SUBAPPLICATION Uebung_206b_AX (* Interlock: ILOCK_T_FF_SR_AX (2 gegenseitig verriegelte Toggle-Flip-Flops via Adapter-Kette, zusaetzlich direktes Set/Reset auf FF1) *)
  (* Standard: 61499-2; Description: Copyright (c) 2026 Meisterschulen am Ostbahnhof This program and the accompanying materials are made available under the terms of the Eclipse Public License 2.0 which is available at https://www.eclipse.org/legal/epl-2.0/ SPDX-License-Identifier: EPL-2.0 *)
  (* Version 1.0, 2026-09-07, Franz Höpfinger, Meisterschulen am Ostbahnhof, initial API and implementation and/or initial documentation - TRAINING_GAPS.md Punkt 7 *)
  PACKAGE Uebungen;
  IMPORT logiBUS::io::DI::logiBUS_DI::Input_I1;
  IMPORT logiBUS::io::DI::logiBUS_DI::Input_I2;
  IMPORT logiBUS::io::DI::logiBUS_DI::Input_I3;
  IMPORT logiBUS::io::DI::logiBUS_DI::Input_I4;
  IMPORT logiBUS::io::DI::logiBUS_DI_Events::BUTTON_SINGLE_CLICK;
  IMPORT logiBUS::io::DQ::logiBUS_DO::Output_Q1;
  IMPORT logiBUS::io::DQ::logiBUS_DO::Output_Q2;
  (* Documentation:
  ILOCK_T_FF_SR_AX: Verriegelbares Toggle-Flip-Flop mit direktem Set/Reset
   Letzter bisher ungenutzter ILOCK-Typ (siehe ILOCK_README.md, "Nicht in Übungen verwendet"). Erweitert ILOCK_T_FF_AX (siehe Uebung_206_AX) um zwei zusätzliche EventInputs S/R: der Ausgang lässt sich nicht nur per CLK togglen, sondern auch direkt setzen/rücksetzen - beides wirkt über dieselbe ILOCK_IN/ILOCK_OUT-Adapterkette gegenseitig verriegelnd auf die anderen Kettenglieder.
   Funktionsbeschreibung
    - Zwei ILOCK_T_FF_SR_AX-Instanzen sind über ILOCK_T_FF_SR_1.ILOCK_OUT → ILOCK_T_FF_SR_2.ILOCK_IN verkettet - genau wie bei ILOCK_T_FF_AX.
   - FF1 hat zusätzlich eigene Set-/Reset-Taster (I3/I4). Ein direktes Set auf FF1 verriegelt FF2 genauso, als hätte man FF1 per CLK eingeschaltet - die Verriegelungskette unterscheidet nicht, ob ein Zustandswechsel durch Toggle oder durch direktes S/R ausgelöst wurde.
    Arbeitsauftrag
   Testen Sie: I1 (CLK FF1) klicken → Q1 EIN, Q2 automatisch AUS (wie in 206). I3 (Set FF1) klicken → dasselbe Ergebnis, aber ohne Toggle - Q1 ist danach garantiert EIN, unabhängig vom vorherigen Zustand. I4 (Reset FF1) klicken → Q1 AUS (Q2 bleibt unverändert, da Reset kein Verriegelungssignal an die Kette sendet - vergleichen Sie das Verhalten von CLK/S vs. R im Baustein-Netzwerk von ILOCK_T_FF_SR_AX).
  *)
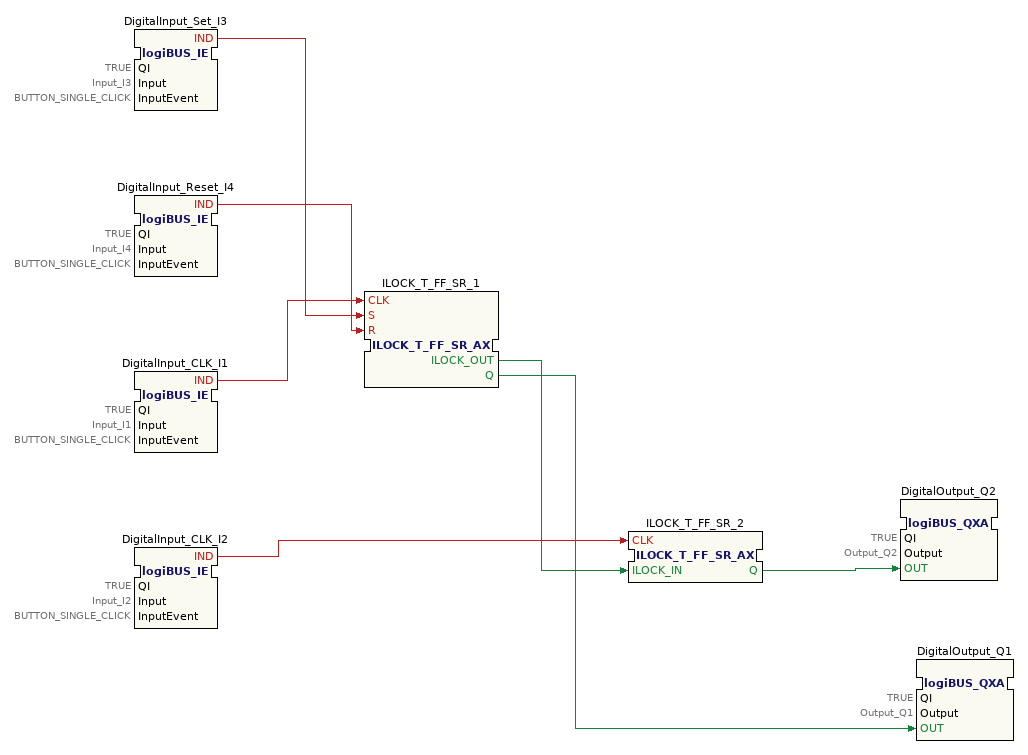
  (* Wie Uebung_206_AX (ILOCK_T_FF_AX), aber ILOCK_T_FF_SR_AX statt ILOCK_T_FF_AX: zusaetzlich zum CLK-Toggle gibt es je Instanz direkte S/R-Eingaenge. Hier nur an FF1 gezeigt (I3=Set, I4=Reset) - Set/Reset auf FF1 loest ueber die Adapter-Kette (ILOCK_OUT->ILOCK_IN) dieselbe gegenseitige Verriegelung aus wie ein CLK-Toggle: wird FF1 gesetzt, wird FF2 automatisch zurueckgesetzt und umgekehrt. *)
  FBS
    DigitalInput_CLK_I1 : logiBUS::io::DI::logiBUS_IE(QI := TRUE, Input := Input_I1, InputEvent := BUTTON_SINGLE_CLICK);
    DigitalInput_Set_I3 : logiBUS::io::DI::logiBUS_IE(QI := TRUE, Input := Input_I3, InputEvent := BUTTON_SINGLE_CLICK);
    DigitalInput_Reset_I4 : logiBUS::io::DI::logiBUS_IE(QI := TRUE, Input := Input_I4, InputEvent := BUTTON_SINGLE_CLICK);
    DigitalInput_CLK_I2 : logiBUS::io::DI::logiBUS_IE(QI := TRUE, Input := Input_I2, InputEvent := BUTTON_SINGLE_CLICK);
    ILOCK_T_FF_SR_1 : logiBUS::signalprocessing::interlock::ILOCK_T_FF_SR_AX;
    ILOCK_T_FF_SR_2 : logiBUS::signalprocessing::interlock::ILOCK_T_FF_SR_AX;
    DigitalOutput_Q1 : logiBUS::io::DQ::logiBUS_QXA(QI := TRUE, Output := Output_Q1);
    DigitalOutput_Q2 : logiBUS::io::DQ::logiBUS_QXA(QI := TRUE, Output := Output_Q2);
  END_FBS
  EVENT_CONNECTIONS
    DigitalInput_CLK_I1.IND TO ILOCK_T_FF_SR_1.CLK;
    DigitalInput_Set_I3.IND TO ILOCK_T_FF_SR_1.S;
    DigitalInput_Reset_I4.IND TO ILOCK_T_FF_SR_1.R;
    DigitalInput_CLK_I2.IND TO ILOCK_T_FF_SR_2.CLK;
  END_CONNECTIONS
  ADAPTER_CONNECTIONS
    ILOCK_T_FF_SR_1.ILOCK_OUT TO ILOCK_T_FF_SR_2.ILOCK_IN;
    ILOCK_T_FF_SR_1.Q TO DigitalOutput_Q1.OUT;
    ILOCK_T_FF_SR_2.Q TO DigitalOutput_Q2.OUT;
  END_CONNECTIONS
END_SUBAPPLICATION
